(* PLC project branches, plcc plcc tests 1 *)
(* stored: creationDateTime 2026-09-27T00:00:00 *)

FUNCTION_BLOCK Branches
  VAR_INPUT
    A : BOOL;
    B : BOOL;
    C : BOOL;
    D : BOOL;
    E : BOOL;
    F : BOOL;
    G : BOOL;
    H : BOOL;
  END_VAR
  VAR_OUTPUT
    Out1 : BOOL;
    X : BOOL;
    Y : BOOL;
    Z : BOOL;
    W : BOOL;
  END_VAR

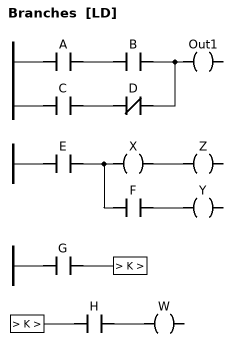
(* LD diagram, written out as Structured Text *)
Out1 := A AND B OR C AND NOT D;
X := E;
Z := E;
Y := E AND F;
W := G AND H;
END_FUNCTION_BLOCK

PROGRAM Main
  VAR
    br : Branches;
  END_VAR

br();
END_PROGRAM
